PROGRAM z_DRAIN

(*-------------------------------------------------------------------------------------------------------*)
(*v015 Ev. Vaciado Gravidad*)
MC._05_DRAIN.v015_Grv.xOpen:= F_VACIADO.z_DrainValveGrv;

(*-------------------------------------------------------------------------------------------------------*)
(*v016 Ev. Vaciado 2 Gravidad*)


(*-------------------------------------------------------------------------------------------------------*)
(*v017 Ev. Vaciado Con Bomba*)
MC._05_DRAIN.v017_Pump.xOpen:= F_VACIADO.z_DrainValvePump;

END_PROGRAM

(* stored: Version 1.1.0.1, ProductVersion 3.1.4024.10
   POU z_DRAIN: Id {d3bb7290-da44-4f84-8764-07165e0e713d}, SpecialFunc None *)
